{attribute 'linkalways'} 
{attribute 'no_explicit_call' := 'This FB is a CLASS and must be accessed using methods or properties'}
{attribute 'enable_dynamic_creation'}
FUNCTION_BLOCK FINAL SEL_WORD EXTENDS Node
VAR
	g : _BOOL(FALSE);
	in1 : _WORD(0);
	in2 : _WORD(0);
	out : _WORD(0);
END_VAR

METHOD PUBLIC Clone : I_Node
VAR
	pNode : POINTER TO SEL_WORD;
END_VAR
pNode := __NEW(SEL_WORD);
Clone := pNode^;
END_METHOD

METHOD FB_init : BOOL
VAR_INPUT
	bInitRetains : BOOL; // if TRUE, the retain variables are initialized (warm start / cold start)
	bInCopyCode : BOOL;  // if TRUE, the instance afterwards gets moved into the copy code (online change)
END_VAR
AddInput('g',THIS^.g);
AddInput('in1',THIS^.in1);
AddInput('in2',THIS^.in2);
AddOutput('out', THIS^.out);
END_METHOD

METHOD PROTECTED OnExecute
VAR
END_VAR
IF g.value THEN
	out.value := in2.value;
ELSE
	out.value := in1.value;
END_IF
END_METHOD

END_FUNCTION_BLOCK

(* stored: Version 1.1.0.1, ProductVersion 3.1.4024.15
   POU SEL_WORD: Id {2f6b6634-c86f-4659-b19c-5ce4cc03e1ab}, SpecialFunc None
   Folder Constructor: Id {66a09899-6f90-48d0-bbf8-c1afab9d6868}
   Method Clone: Id {589d16a0-065f-457f-beb3-daf1b05bf600}
   Method FB_init: Id {0bf1b136-d019-4a55-a3bc-dd20fe2ba8f8}
   Method OnExecute: Id {6df77cbe-4a47-4380-ba01-34747adc918b} *)
